{attribute addProperty BoxType "EPP1322-0001-0017"}
{attribute addProperty Id "A_0021_EPP1332_0001_0016A_0021_EPP1332_0001_0016_0CFFDA602816352"}
{attribute addProperty CRC "3605475596"}
{attribute addProperty SizeInBites "2816"}
{attribute addProperty SizeInBytes "352"}
TYPE A_0020_EPP1322_0001_0017_D6E7310C EXTENDS EPP1322_179A0949 :
STRUCT
	{attribute addProperty Name "A_0021_EPP1332_0001_0016"}
	A_0021_EPP1332_0001_0016 : A_0021_EPP1332_0001_0016_0CFFDA60;
END_STRUCT
END_TYPE

(* stored: Version 1.2.0.0, ProductVersion 3.1.4024.9
   DUT A_0020_EPP1322_0001_0017_D6E7310C: Id {b730e799-97ec-46ba-9fbc-89518deb335d} *)
